(* IEC 61131-3 sources: rk/stdlib (part 4) *)

(* ---- Strings.st ---- *)
/*
String functions.

A `STRING` holds UTF-8 text, and its length is a number of bytes. The
functions here come in two families.

`LEN`, `FIND`, `LEFT`, `RIGHT`, `MID`, `INSERT`, `DELETE` and `REPLACE` count
bytes. They are the fast ones, and on ASCII text a byte is a character. On
other text a byte position can fall inside a character, and slicing there
yields a string that is not valid UTF-8.

The `CHAR_` functions count characters and never split one. A character is
one well-formed UTF-8 sequence. A byte that belongs to none counts as a
character on its own, its Latin-1 code point, like `CHAR#'$E9'`.

Positions start at 1 in both families. A function that returns a `STRING`
returns up to 255 bytes, and cuts a longer result there. It is also cut,
without an error, when it does not fit where it is stored.
*/
NAMESPACE Std.Strings

	/* Returns the length of `IN`, in bytes.

	   This is not the number of characters: `LEN('café')` is 5, because `é`
	   takes two bytes. See [Std.Strings.CHAR_COUNT] for that.

	   The length is stored with the string, so this does not scan it.

	   # Examples

	   ```iecst
	   n := LEN('hello');  // 5
	   n := LEN('');       // 0
	   ```
	*/
	FUNCTION LEN: UDINT
		VAR_INPUT
			IN: STRING[255];
		END_VAR
		{wasm 'str.byte_len' (params IN) (result LEN)}
	END_FUNCTION

	/* Returns `TRUE` if `IN` is well-formed UTF-8.

	   Text that comes from outside the program, such as a host import or a
	   fieldbus frame, may not be. Check it before slicing it by bytes.

	   # Examples

	   ```iecst
	   ok := IS_UTF8('café');  // TRUE
	   ok := IS_UTF8('$E9');   // FALSE, a lone Latin-1 byte
	   ```
	*/
	FUNCTION IS_UTF8: BOOL
		VAR_INPUT
			IN: STRING[255];
		END_VAR
		{wasm 'str.is_utf8' (params IN) (result IS_UTF8)}
	END_FUNCTION

	/* Returns the byte position of the first occurrence of `IN2` in
	   `IN1`, or 0 if there is none.

	   Positions start at 1. An empty `IN2` is found at position 1.

	   To look for a single `CHAR`, convert it with [Std.Convert.CHAR_TO_STRING].

	   # Examples

	   ```iecst
	   p := FIND('hello world', 'world');  // 7
	   p := FIND('hello world', 'xyz');    // 0
	   ```
	*/
	FUNCTION FIND: UDINT
		VAR_INPUT
			IN1: STRING[255];
			IN2: STRING[255];
		END_VAR
		{wasm 'str.byte_find' (params IN1 IN2) (result FIND)}
	END_FUNCTION

	/* Returns its inputs one after the other, from two inputs up to eight.

	   To append a single `CHAR`, convert it with [Std.Convert.CHAR_TO_STRING].

	   # Examples

	   ```iecst
	   s := CONCAT('hello ', 'world');  // 'hello world'
	   s := CONCAT('a', 'b', 'c');      // 'abc'
	   ```
	*/
	FUNCTION CONCAT: STRING[255]
		VAR_INPUT
			IN1: STRING[255];
			IN2: STRING[255];
		END_VAR
		{wasm 'str.concat' (params IN1 IN2) (result CONCAT)}
	END_FUNCTION

	FUNCTION CONCAT: STRING[255]
		VAR_INPUT
			IN1: STRING[255];
			IN2: STRING[255];
			IN3: STRING[255];
		END_VAR

		CONCAT := CONCAT(IN1, IN2);
		CONCAT := CONCAT(CONCAT, IN3);
	END_FUNCTION

	FUNCTION CONCAT: STRING[255]
		VAR_INPUT
			IN1: STRING[255];
			IN2: STRING[255];
			IN3: STRING[255];
			IN4: STRING[255];
		END_VAR

		CONCAT := CONCAT(IN1, IN2);
		CONCAT := CONCAT(CONCAT, IN3);
		CONCAT := CONCAT(CONCAT, IN4);
	END_FUNCTION

	FUNCTION CONCAT: STRING[255]
		VAR_INPUT
			IN1: STRING[255];
			IN2: STRING[255];
			IN3: STRING[255];
			IN4: STRING[255];
			IN5: STRING[255];
		END_VAR

		CONCAT := CONCAT(IN1, IN2);
		CONCAT := CONCAT(CONCAT, IN3);
		CONCAT := CONCAT(CONCAT, IN4);
		CONCAT := CONCAT(CONCAT, IN5);
	END_FUNCTION

	FUNCTION CONCAT: STRING[255]
		VAR_INPUT
			IN1: STRING[255];
			IN2: STRING[255];
			IN3: STRING[255];
			IN4: STRING[255];
			IN5: STRING[255];
			IN6: STRING[255];
		END_VAR

		CONCAT := CONCAT(IN1, IN2);
		CONCAT := CONCAT(CONCAT, IN3);
		CONCAT := CONCAT(CONCAT, IN4);
		CONCAT := CONCAT(CONCAT, IN5);
		CONCAT := CONCAT(CONCAT, IN6);
	END_FUNCTION

	FUNCTION CONCAT: STRING[255]
		VAR_INPUT
			IN1: STRING[255];
			IN2: STRING[255];
			IN3: STRING[255];
			IN4: STRING[255];
			IN5: STRING[255];
			IN6: STRING[255];
			IN7: STRING[255];
		END_VAR

		CONCAT := CONCAT(IN1, IN2);
		CONCAT := CONCAT(CONCAT, IN3);
		CONCAT := CONCAT(CONCAT, IN4);
		CONCAT := CONCAT(CONCAT, IN5);
		CONCAT := CONCAT(CONCAT, IN6);
		CONCAT := CONCAT(CONCAT, IN7);
	END_FUNCTION

	FUNCTION CONCAT: STRING[255]
		VAR_INPUT
			IN1: STRING[255];
			IN2: STRING[255];
			IN3: STRING[255];
			IN4: STRING[255];
			IN5: STRING[255];
			IN6: STRING[255];
			IN7: STRING[255];
			IN8: STRING[255];
		END_VAR

		CONCAT := CONCAT(IN1, IN2);
		CONCAT := CONCAT(CONCAT, IN3);
		CONCAT := CONCAT(CONCAT, IN4);
		CONCAT := CONCAT(CONCAT, IN5);
		CONCAT := CONCAT(CONCAT, IN6);
		CONCAT := CONCAT(CONCAT, IN7);
		CONCAT := CONCAT(CONCAT, IN8);
	END_FUNCTION

	/* Returns the first `L` bytes of `IN`.

	   Returns all of `IN` when `L` is greater than its length.

	   # Examples

	   ```iecst
	   s := LEFT('hello world', 5);  // 'hello'
	   s := LEFT('hi', 10);          // 'hi'
	   ```
	*/
	FUNCTION LEFT: STRING[255]
		VAR_INPUT
			IN: STRING[255];
			L: UDINT;
		END_VAR
		{wasm 'str.byte_left' (params IN L) (result LEFT)}
	END_FUNCTION

	/* Returns the last `L` bytes of `IN`.

	   Returns all of `IN` when `L` is greater than its length.

	   # Examples

	   ```iecst
	   s := RIGHT('hello world', 5);  // 'world'
	   s := RIGHT('hi', 10);          // 'hi'
	   ```
	*/
	FUNCTION RIGHT: STRING[255]
		VAR_INPUT
			IN: STRING[255];
			L: UDINT;
		END_VAR
		{wasm 'str.byte_right' (params IN L) (result RIGHT)}
	END_FUNCTION

	/* Returns `L` bytes of `IN`, starting at byte position `P`.

	   Returns fewer when `IN` ends first, and an empty string when `P` is 0 or
	   past the end.

	   # Examples

	   ```iecst
	   s := MID('hello world', 5, 7);  // 'world'
	   s := MID('hello', 10, 3);       // 'llo'
	   s := MID('hello', 3, 10);       // ''
	   ```
	*/
	FUNCTION MID: STRING[255]
		VAR_INPUT
			IN: STRING[255];
			L: UDINT;
			P: UDINT;
		END_VAR
		{wasm 'str.byte_mid' (params IN L P) (result MID)}
	END_FUNCTION

	/* Returns `IN1` with `IN2` inserted after byte position `P`.

	   A `P` of 0 inserts at the front.

	   To insert a single `CHAR`, convert it with [Std.Convert.CHAR_TO_STRING].

	   # Examples

	   ```iecst
	   s := INSERT('helloworld', 'XX', 5);  // 'helloXXworld'
	   s := INSERT('world', 'hello ', 0);   // 'hello world'
	   ```
	*/
	FUNCTION INSERT: STRING[255]
		VAR_INPUT
			IN1: STRING[255];
			IN2: STRING[255];
			P: UDINT;
		END_VAR
		{wasm 'str.byte_insert' (params IN1 IN2 P) (result INSERT)}
	END_FUNCTION

	/* Returns `IN` without the `L` bytes that start at byte position `P`.

	   Removes fewer when `IN` ends first, and nothing when `P` is past the end.

	   # Examples

	   ```iecst
	   s := DELETE('hello world', 6, 6);  // 'hello'
	   s := DELETE('hello', 10, 3);       // 'he'
	   s := DELETE('hello', 3, 10);       // 'hello'
	   ```
	*/
	FUNCTION DELETE: STRING[255]
		VAR_INPUT
			IN: STRING[255];
			L: UDINT;
			P: UDINT;
		END_VAR
		{wasm 'str.byte_delete' (params IN L P) (result DELETE)}
	END_FUNCTION

	/* Returns `IN1` with the `L` bytes that start at byte position `P` replaced
	   by `IN2`.

	   `IN2` does not have to be `L` bytes long.

	   To replace with a single `CHAR`, convert it with [Std.Convert.CHAR_TO_STRING].

	   # Examples

	   ```iecst
	   s := REPLACE('hello world', 'there', 5, 7);  // 'hello there'
	   s := REPLACE('hello world', '!', 5, 7);      // 'hello !'
	   ```
	*/
	FUNCTION REPLACE: STRING[255]
		VAR_INPUT
			IN1: STRING[255];
			IN2: STRING[255];
			L: UDINT;
			P: UDINT;
		END_VAR
		{wasm 'str.byte_replace' (params IN1 IN2 L P) (result REPLACE)}
	END_FUNCTION

	/* Returns the number of characters in `IN`.

	   # Examples

	   ```iecst
	   n := CHAR_COUNT('café');    // 4, where LEN returns 5
	   n := CHAR_COUNT('日本語');  // 3, where LEN returns 9
	   ```
	*/
	FUNCTION CHAR_COUNT: UDINT
		VAR_INPUT
			IN: STRING[255];
		END_VAR
		{wasm 'str.char_count' (params IN) (result CHAR_COUNT)}
	END_FUNCTION

	/* Returns the character at position `P` of `IN`.

	   Returns `CHAR#'$00'` when `P` is 0 or past the end.

	   # Examples

	   ```iecst
	   c := CHAR_AT('café', 4);  // CHAR#'é'
	   c := CHAR_AT('abc', 4);   // CHAR#'$00'
	   ```
	*/
	FUNCTION CHAR_AT: CHAR
		VAR_INPUT
			IN: STRING[255];
			P: UDINT;
		END_VAR
		{wasm 'str.char_at' (params IN P) (result CHAR_AT)}
	END_FUNCTION

	/* Returns the character position of the first occurrence of `IN2` in
	   `IN1`, or 0 if there is none.

	   An empty `IN2` is found at position 1, as with [Std.Strings.FIND].

	   # Examples

	   ```iecst
	   p := CHAR_FIND('日本語', '語');  // 3, where FIND returns 7
	   p := CHAR_FIND('abc', 'x');      // 0
	   ```
	*/
	FUNCTION CHAR_FIND: UDINT
		VAR_INPUT
			IN1: STRING[255];
			IN2: STRING[255];
		END_VAR
		{wasm 'str.char_find' (params IN1 IN2) (result CHAR_FIND)}
	END_FUNCTION

	/* Returns the first `L` characters of `IN`.

	   Returns all of `IN` when `L` is greater than its character count.

	   # Examples

	   ```iecst
	   s := CHAR_LEFT('café', 3);   // 'caf'
	   s := CHAR_LEFT('café', 10);  // 'café'
	   ```
	*/
	FUNCTION CHAR_LEFT: STRING[255]
		VAR_INPUT
			IN: STRING[255];
			L: UDINT;
		END_VAR
		{wasm 'str.char_left' (params IN L) (result CHAR_LEFT)}
	END_FUNCTION

	/* Returns the last `L` characters of `IN`.

	   Returns all of `IN` when `L` is greater than its character count.

	   # Examples

	   ```iecst
	   s := CHAR_RIGHT('日本語', 2);  // '本語'
	   s := CHAR_RIGHT('café', 1);    // 'é'
	   ```
	*/
	FUNCTION CHAR_RIGHT: STRING[255]
		VAR_INPUT
			IN: STRING[255];
			L: UDINT;
		END_VAR
		{wasm 'str.char_right' (params IN L) (result CHAR_RIGHT)}
	END_FUNCTION

	/* Returns `L` characters of `IN`, starting at character position `P`.

	   Returns fewer when `IN` ends first, and an empty string when `P` is 0 or
	   past the end.

	   # Examples

	   ```iecst
	   s := CHAR_MID('café', 2, 3);    // 'fé'
	   s := CHAR_MID('日本語', 1, 2);  // '本'
	   ```
	*/
	FUNCTION CHAR_MID: STRING[255]
		VAR_INPUT
			IN: STRING[255];
			L: UDINT;
			P: UDINT;
		END_VAR
		{wasm 'str.char_mid' (params IN L P) (result CHAR_MID)}
	END_FUNCTION

	/* Returns `IN1` with `IN2` inserted after character position `P`.

	   A `P` of 0 inserts at the front, and a `P` past the end appends.

	   # Examples

	   ```iecst
	   s := CHAR_INSERT('caf', 'é', 3);    // 'café'
	   s := CHAR_INSERT('abc', 'X', 0);    // 'Xabc'
	   s := CHAR_INSERT('café', 'X', 99);  // 'caféX'
	   ```
	*/
	FUNCTION CHAR_INSERT: STRING[255]
		VAR_INPUT
			IN1: STRING[255];
			IN2: STRING[255];
			P: UDINT;
		END_VAR
		{wasm 'str.char_insert' (params IN1 IN2 P) (result CHAR_INSERT)}
	END_FUNCTION

	/* Returns `IN` without the `L` characters that start at character
	   position `P`.

	   Returns `IN` unchanged when `P` is 0 or past the end.

	   # Examples

	   ```iecst
	   s := CHAR_DELETE('日本語', 1, 2);  // '日語'
	   s := CHAR_DELETE('café', 1, 5);    // 'café'
	   ```
	*/
	FUNCTION CHAR_DELETE: STRING[255]
		VAR_INPUT
			IN: STRING[255];
			L: UDINT;
			P: UDINT;
		END_VAR
		{wasm 'str.char_delete' (params IN L P) (result CHAR_DELETE)}
	END_FUNCTION

	/* Returns `IN1` with the `L` characters that start at character position
	   `P` replaced by `IN2`.

	   Returns `IN1` unchanged when `P` is 0 or past the end.

	   # Examples

	   ```iecst
	   s := CHAR_REPLACE('café', 'e', 1, 4);    // 'cafe'
	   s := CHAR_REPLACE('日本語', 'X', 2, 1);  // 'X語'
	   ```
	*/
	FUNCTION CHAR_REPLACE: STRING[255]
		VAR_INPUT
			IN1: STRING[255];
			IN2: STRING[255];
			L: UDINT;
			P: UDINT;
		END_VAR
		{wasm 'str.char_replace' (params IN1 IN2 L P) (result CHAR_REPLACE)}
	END_FUNCTION

	NAMESPACE Test
		USING Std.Unit
		USING Std.Convert

		{test}
		FUNCTION test_len_ascii
			ASSERT(LEN('hello') = 5);
		END_FUNCTION

		{test}
		FUNCTION test_len_empty
			ASSERT(LEN('') = 0);
		END_FUNCTION

		{test}
		FUNCTION test_len_counts_utf8_bytes
			ASSERT(LEN('café') = 5 AND LEN('€') = 3 AND LEN('中文') = 6);
			ASSERT(IS_UTF8('café') AND IS_UTF8('中文'));
			{allow 'latin1-escape'}
			ASSERT(LEN('$E9') = 1 AND NOT IS_UTF8('$E9'));
		END_FUNCTION

		{test}
		FUNCTION test_is_utf8_ascii
			ASSERT(IS_UTF8('hello'));
		END_FUNCTION

		{test}
		FUNCTION test_is_utf8_empty
			ASSERT(IS_UTF8(''));
		END_FUNCTION

		{test}
		FUNCTION test_find_present
			ASSERT(FIND('hello world', 'world') = 7);
		END_FUNCTION

		{test}
		FUNCTION test_find_at_start
			ASSERT(FIND('hello world', 'hello') = 1);
		END_FUNCTION

		{test}
		FUNCTION test_find_missing
			ASSERT(FIND('hello world', 'xyz') = 0);
		END_FUNCTION

		{test}
		FUNCTION test_find_empty_needle
			ASSERT(FIND('hello', '') = 1);
		END_FUNCTION

		{test}
		FUNCTION test_find_needle_longer_than_haystack
			ASSERT(FIND('hi', 'hello') = 0);
		END_FUNCTION

		{test}
		FUNCTION test_concat_basic
			VAR result: STRING; END_VAR
			result := CONCAT('hello ', 'world');
			ASSERT(LEN(result) = 11);
			ASSERT(FIND(result, 'hello world') = 1);
		END_FUNCTION

		{test}
		FUNCTION test_concat_empty_left
			VAR result: STRING; END_VAR
			result := CONCAT('', 'world');
			ASSERT(LEN(result) = 5);
		END_FUNCTION

		{test}
		FUNCTION test_concat_empty_right
			VAR result: STRING; END_VAR
			result := CONCAT('hello', '');
			ASSERT(LEN(result) = 5);
		END_FUNCTION

		// A result holds up to 255 bytes, not the default 80: what does not
		// fit is cut where it is stored.
		{test}
		FUNCTION test_concat_keeps_more_than_80_bytes
			VAR
				a: STRING[100] := '0123456789012345678901234567890123456789012345678901234567890123456789012345678901234567890123456789';
				result: STRING[200];
			END_VAR
			result := CONCAT(a, a);
			ASSERT(LEN(result) = 200);
		END_FUNCTION

		{test}
		FUNCTION test_a_result_is_cut_at_255_bytes
			VAR
				a: STRING[200] := '01234567890123456789012345678901234567890123456789012345678901234567890123456789012345678901234567890123456789012345678901234567890123456789012345678901234567890123456789012345678901234567890123456789';
				result: STRING[300];
			END_VAR
			result := CONCAT(a, a);
			// LEN reads 255 bytes at most: the result holds 255.
			{allow 'string-truncation'}
			ASSERT(LEN(result) = 255);
		END_FUNCTION

		{test}
		FUNCTION test_delete_one_byte_of_a_100_byte_string
			VAR s: STRING[200] := '0123456789012345678901234567890123456789012345678901234567890123456789012345678901234567890123456789'; END_VAR
			s := DELETE(s, 1, 1);
			ASSERT(LEN(s) = 99);
		END_FUNCTION

		{test}
		FUNCTION test_left_basic
			VAR result: STRING; END_VAR
			result := LEFT('hello world', 5);
			ASSERT(LEN(result) = 5);
			ASSERT(FIND(result, 'hello') = 1);
		END_FUNCTION

		{test}
		FUNCTION test_left_n_exceeds_length
			VAR result: STRING; END_VAR
			result := LEFT('hi', 10);
			ASSERT(LEN(result) = 2);
		END_FUNCTION

		{test}
		FUNCTION test_right_basic
			VAR result: STRING; END_VAR
			result := RIGHT('hello world', 5);
			ASSERT(LEN(result) = 5);
			ASSERT(FIND(result, 'world') = 1);
		END_FUNCTION

		{test}
		FUNCTION test_mid_basic
			VAR result: STRING; END_VAR
			// 'world' starts at byte 7, 5 chars
			result := MID('hello world', 5, 7);
			ASSERT(LEN(result) = 5);
			ASSERT(FIND(result, 'world') = 1);
		END_FUNCTION

		{test}
		FUNCTION test_mid_p_zero
			VAR result: STRING; END_VAR
			result := MID('hello', 3, 0);
			ASSERT(LEN(result) = 0);
		END_FUNCTION

		{test}
		FUNCTION test_insert_middle
			VAR result: STRING; END_VAR
			// Insert 'XX' after byte 5 of 'helloworld' → 'helloXXworld'
			result := INSERT('helloworld', 'XX', 5);
			ASSERT(LEN(result) = 12);
			ASSERT(FIND(result, 'helloXXworld') = 1);
		END_FUNCTION

		{test}
		FUNCTION test_insert_front
			VAR result: STRING; END_VAR
			result := INSERT('world', 'hello ', 0);
			ASSERT(LEN(result) = 11);
			ASSERT(FIND(result, 'hello world') = 1);
		END_FUNCTION

		{test}
		FUNCTION test_delete_basic
			VAR result: STRING; END_VAR
			// Delete 6 bytes starting at byte 6 of 'hello world' → 'hello'
			result := DELETE('hello world', 6, 6);
			ASSERT(LEN(result) = 5);
			ASSERT(FIND(result, 'hello') = 1);
		END_FUNCTION

		{test}
		FUNCTION test_replace_basic
			VAR result: STRING; END_VAR
			// Replace 5 bytes at byte 7 of 'hello world' with 'there'
			result := REPLACE('hello world', 'there', 5, 7);
			ASSERT(LEN(result) = 11);
			ASSERT(FIND(result, 'hello there') = 1);
		END_FUNCTION

		{test}
		FUNCTION test_concat_nested_binary
			// Independent inner CONCATs feeding an outer CONCAT: each
			// inner result must survive long enough for the outer to read
			// it. With per-call-site scratch slots: 'xxyyzzww'.
			VAR result: STRING; END_VAR
			result := CONCAT(CONCAT('xx', 'yy'), CONCAT('zz', 'ww'));
			ASSERT(LEN(result) = 8);
			ASSERT(FIND(result, 'xxyyzzww') = 1);
		END_FUNCTION

		{test}
		FUNCTION test_concat_nested_left_arg
			// Inner result used as outer's first arg.
			VAR result: STRING; END_VAR
			result := CONCAT(CONCAT('ab', 'cd'), 'ef');
			ASSERT(LEN(result) = 6);
			ASSERT(FIND(result, 'abcdef') = 1);
		END_FUNCTION

		{test}
		FUNCTION test_left_inside_concat
			VAR result: STRING; END_VAR
			result := CONCAT(LEFT('hello world', 5), '!');
			ASSERT(LEN(result) = 6);
			ASSERT(FIND(result, 'hello!') = 1);
		END_FUNCTION

		/* CHAR-as-string usage: explicit conversion via
		   `Std.Convert.CHAR_TO_STRING`. CHAR is an i32 code point at
		   the WASM ABI; CONCAT/INSERT/REPLACE/FIND all take STRING args,
		   so users wrap CHAR values explicitly. */

		{test}
		FUNCTION test_concat_char_literal_right
			VAR result: STRING; END_VAR
			result := CONCAT('hello', CHAR_TO_STRING(CHAR#'!'));
			ASSERT(LEN(result) = 6);
			ASSERT(FIND(result, 'hello!') = 1);
		END_FUNCTION

		{test}
		FUNCTION test_concat_char_literal_left
			VAR result: STRING; END_VAR
			result := CONCAT(CHAR_TO_STRING(CHAR#'>'), ' message');
			ASSERT(LEN(result) = 9);
			ASSERT(FIND(result, '> message') = 1);
		END_FUNCTION

		{test}
		FUNCTION test_find_char_literal_needle
			ASSERT(FIND('hello', CHAR_TO_STRING(CHAR#'l')) = 3);
		END_FUNCTION

		{test}
		FUNCTION test_insert_char_literal
			VAR result: STRING; END_VAR
			result := INSERT('helloworld', CHAR_TO_STRING(CHAR#' '), 5);
			ASSERT(LEN(result) = 11);
			ASSERT(FIND(result, 'hello world') = 1);
		END_FUNCTION

		{test}
		FUNCTION test_replace_char_literal
			VAR result: STRING; END_VAR
			// Replace 5 bytes at byte 7 of 'hello world' with the single CHAR '!'.
			result := REPLACE('hello world', CHAR_TO_STRING(CHAR#'!'), 5, 7);
			ASSERT(LEN(result) = 7);
			ASSERT(FIND(result, 'hello !') = 1);
		END_FUNCTION

		{test}
		FUNCTION test_concat_char_var
			VAR
				bang: CHAR := CHAR#'!';
				result: STRING;
			END_VAR
			result := CONCAT('hello', CHAR_TO_STRING(bang));
			ASSERT(LEN(result) = 6);
			ASSERT(FIND(result, 'hello!') = 1);
		END_FUNCTION

		{test}
		FUNCTION test_find_char_var
			VAR
				needle: CHAR := CHAR#'l';
			END_VAR
			ASSERT(FIND('hello', CHAR_TO_STRING(needle)) = 3);
		END_FUNCTION

		{test}
		FUNCTION test_concat_char_var_left
			VAR
				prefix: CHAR := CHAR#'>';
				result: STRING;
			END_VAR
			result := CONCAT(CHAR_TO_STRING(prefix), ' message');
			ASSERT(LEN(result) = 9);
			ASSERT(FIND(result, '> message') = 1);
		END_FUNCTION

		{test}
		FUNCTION test_concat_two_char_vars
			// Two nested CHAR_TO_STRING calls: each must get its own
			// per-call-site scratch slot, the second mustn't clobber the
			// first before the outer CONCAT reads them.
			VAR
				a: CHAR := CHAR#'a';
				b: CHAR := CHAR#'b';
				result: STRING;
			END_VAR
			result := CONCAT(CHAR_TO_STRING(a), CHAR_TO_STRING(b));
			ASSERT(LEN(result) = 2);
			ASSERT(FIND(result, 'ab') = 1);
		END_FUNCTION

		// --- return-slot aliasing: results copied into locals must survive
		// LATER producer calls (the dangerous scenario of a shared static
		// return slot), and self-argument accumulation must not corrupt ---

		{test}
		FUNCTION test_result_survives_later_producer_call
			VAR
				first, second: STRING;
			END_VAR
			first := CONCAT('aa', 'bb');
			second := CONCAT('cc', 'dd');
			ASSERT(FIND(first, 'aabb') = 1, 'earlier result must survive a later producer call');
			ASSERT(FIND(second, 'ccdd') = 1, 'later result is correct too');
		END_FUNCTION

		{test}
		FUNCTION test_concat_self_accumulation
			VAR
				s: STRING;
				i: INT;
			END_VAR
			s := 'x';
			FOR i := 1 TO 4 DO
				s := CONCAT(s, 'y');
			END_FOR;
			ASSERT(LEN(s) = 5, 'x + 4 accumulated y');
			ASSERT(FIND(s, 'xyyyy') = 1, 'self-argument CONCAT accumulates correctly');
		END_FUNCTION

		// --- slicer bounds: N/P beyond the string must clamp, not underflow ---

		{test}
		FUNCTION test_right_n_beyond_length
			VAR
				s: STRING;
			END_VAR
			// RIGHT computes len-N internally: N > len must clamp, not
			// underflow to a huge unsigned offset.
			s := RIGHT('hi', 10);
			ASSERT(LEN(s) = 2, 'RIGHT with N beyond length returns the whole string');
			ASSERT(FIND(s, 'hi') = 1, 'content intact');
		END_FUNCTION

		{test}
		FUNCTION test_mid_beyond_length
			VAR
				s: STRING;
			END_VAR
			s := MID('hello', 10, 3);
			ASSERT(LEN(s) = 3, 'MID clamps L to the remaining chars');
			s := MID('hello', 3, 10);
			ASSERT(LEN(s) = 0, 'MID with P beyond length yields empty');
		END_FUNCTION

		{test}
		FUNCTION test_delete_beyond_length
			VAR
				s: STRING;
			END_VAR
			// Signature is DELETE(S, N, P): delete N chars at position P.
			s := DELETE('hello', 3, 10);
			ASSERT(LEN(s) = 5, 'DELETE at P beyond the end removes nothing');
			s := DELETE('hello', 10, 3);
			ASSERT(LEN(s) = 2, 'DELETE clamps N to the remaining chars (keeps "he")');
			ASSERT(FIND(s, 'he') = 1, 'prefix before P survives');
		END_FUNCTION

		{test}
		FUNCTION test_find_no_match_returns_zero
			ASSERT(FIND('hello', 'xyz') = 0, 'FIND with no match returns 0');
			ASSERT(FIND('', 'a') = 0, 'FIND in empty string returns 0');
		END_FUNCTION

		{test}
		FUNCTION test_len_zero_slices
			VAR
				s: STRING;
			END_VAR
			s := LEFT('hello', 0);
			ASSERT(LEN(s) = 0, 'LEFT L=0 is empty');
			s := MID('hello', 0, 2);
			ASSERT(LEN(s) = 0, 'MID L=0 is empty');
		END_FUNCTION

		// --- STRING comparison operators: =, <>, and lexicographic ordering
		// (byte-wise with length tiebreak). These replace the LEN+FIND idiom
		// for content assertions. ---

		{test}
		FUNCTION test_string_equality_operators
			VAR
				s: STRING := 'START';
			END_VAR
			ASSERT(s = 'START', 'var = literal');
			ASSERT('START' = s, 'literal = var');
			ASSERT(s <> 'STOP', 'not-equal');
			ASSERT_EQ(CONCAT('STA', 'RT'), 'START', 'ASSERT_EQ on a producer result');
			ASSERT_NEQ(CONCAT('a', 'b'), 'ba', 'ASSERT_NEQ on unequal content');
		END_FUNCTION

		{test}
		FUNCTION test_string_ordering_operators
			ASSERT('abc' < 'abd', 'lexicographic less');
			ASSERT('ab' < 'abc', 'shared prefix: shorter is smaller');
			ASSERT('abd' > 'abc', 'greater');
			ASSERT('abc' <= 'abc', 'le on equal');
			ASSERT('abc' >= 'abc', 'ge on equal');
			ASSERT(NOT ('abc' < 'abc'), 'not strictly less than itself');
			ASSERT('' < 'a', 'empty sorts first');
		END_FUNCTION

		{test}
		FUNCTION test_string_equality_after_mutation
			VAR
				s: STRING := 'x';
				i: INT;
			END_VAR
			FOR i := 1 TO 3 DO
				s := CONCAT(s, 'y');
			END_FOR;
			ASSERT_EQ(s, 'xyyy', 'accumulated content compares whole');
		END_FUNCTION

		// Both operands are producer calls: each needs its own scratch
		// buffer. If they shared the one static return slot, the second call
		// would clobber the first and every such comparison would degenerate
		// to comparing a value with itself (silently always equal).
		{test}
		FUNCTION test_string_comparison_between_two_producers
			ASSERT(CONCAT('ab', 'cd') = CONCAT('ab', 'cd'), 'equal producer results compare equal');
			ASSERT(CONCAT('ab', 'cd') <> CONCAT('xy', 'zw'), 'different producer results must not be equal');
			ASSERT(CONCAT('a', 'a') < CONCAT('a', 'b'), 'ordering holds across two producers');
		END_FUNCTION

		// ----- Character-aware twins --------------------------------------
		{test}
		FUNCTION test_char_count_agrees_with_len_on_ascii
			ASSERT(CHAR_COUNT('hello') = 5 AND CHAR_COUNT('') = 0);
			ASSERT(CHAR_COUNT('hello') = LEN('hello'));
		END_FUNCTION

		{test}
		FUNCTION test_char_count_counts_characters_not_bytes
			ASSERT(CHAR_COUNT('café') = 4 AND LEN('café') = 5);
			ASSERT(CHAR_COUNT('日本語') = 3 AND LEN('日本語') = 9);
			{allow 'latin1-escape'}
			ASSERT(CHAR_COUNT('$E9$E9') = 2, 'a stray byte is one character');
		END_FUNCTION

		{test}
		FUNCTION test_char_at_returns_the_character
			ASSERT(CHAR_AT('café', 4) = CHAR#'é' AND CHAR_AT('café', 1) = CHAR#'c');
			ASSERT(CHAR_AT('日本語', 2) = CHAR#'本');
			{allow 'latin1-escape'}
			ASSERT(CHAR_AT('$E9', 1) = CHAR#'é', 'a stray byte reads as its Latin-1 character');
			ASSERT(CHAR_AT('abc', 0) = CHAR#'$00' AND CHAR_AT('abc', 4) = CHAR#'$00');
		END_FUNCTION

		{test}
		FUNCTION test_char_find_counts_characters
			ASSERT(CHAR_FIND('日本語', '語') = 3 AND FIND('日本語', '語') = 7);
			ASSERT(CHAR_FIND('café!', '!') = 5);
			ASSERT(CHAR_FIND('abc', 'x') = 0 AND CHAR_FIND('abc', '') = 1);
		END_FUNCTION

		{test}
		FUNCTION test_char_left_and_right_never_split_a_character
			ASSERT(CHAR_LEFT('café', 4) = 'café' AND CHAR_LEFT('café', 3) = 'caf');
			ASSERT(CHAR_RIGHT('café', 1) = 'é' AND CHAR_RIGHT('日本語', 2) = '本語');
			ASSERT(CHAR_LEFT('café', 10) = 'café' AND CHAR_RIGHT('café', 0) = '');
		END_FUNCTION

		{test}
		FUNCTION test_char_mid_counts_characters
			ASSERT(CHAR_MID('日本語', 1, 2) = '本' AND CHAR_MID('café', 2, 3) = 'fé');
			ASSERT(CHAR_MID('café', 10, 4) = 'é', 'N past the end is clamped');
			ASSERT(CHAR_MID('café', 1, 0) = '' AND CHAR_MID('café', 1, 5) = '');
		END_FUNCTION

		{test}
		FUNCTION test_char_insert_delete_replace_count_characters
			ASSERT(CHAR_INSERT('caf', 'é', 3) = 'café' AND CHAR_INSERT('日語', '本', 1) = '日本語');
			ASSERT(CHAR_INSERT('abc', 'X', 0) = 'Xabc');
			ASSERT(CHAR_DELETE('café', 1, 4) = 'caf' AND CHAR_DELETE('日本語', 1, 2) = '日語');
			ASSERT(CHAR_DELETE('café', 1, 0) = 'café' AND CHAR_DELETE('café', 1, 5) = 'café');
			ASSERT(CHAR_REPLACE('café', 'e', 1, 4) = 'cafe' AND CHAR_REPLACE('日本語', 'X', 2, 1) = 'X語');
			ASSERT(CHAR_REPLACE('café', 'X', 1, 0) = 'café');
		END_FUNCTION

		// A character position past the end maps to a byte position past the
		// end and the byte functions decide: just past and far past must agree.
		{test}
		FUNCTION test_char_positions_past_the_end_agree
			ASSERT(CHAR_MID('café', 2, 5) = CHAR_MID('café', 2, 99) AND CHAR_MID('café', 2, 99) = '');
			ASSERT(CHAR_DELETE('café', 2, 5) = CHAR_DELETE('café', 2, 99) AND CHAR_DELETE('café', 2, 99) = 'café');
			ASSERT(CHAR_REPLACE('café', 'X', 2, 5) = CHAR_REPLACE('café', 'X', 2, 99) AND CHAR_REPLACE('café', 'X', 2, 99) = 'café');
			ASSERT(CHAR_INSERT('café', 'X', 5) = CHAR_INSERT('café', 'X', 99) AND CHAR_INSERT('café', 'X', 99) = 'caféX');
		END_FUNCTION

		// `LEN(s) - k` with k > LEN(s) is an N near 2^32, and `start + n`
		// wrapped on wasm32: MID trapped, DELETE and REPLACE kept the wrong
		// part. CHAR_MID and its kin count N first and never did.
		{test}
		FUNCTION test_mid_delete_replace_with_n_near_the_limit
			ASSERT(MID('hello', UDINT#4294967295, 2) = 'ello', 'MID N = 2^32-1');
			ASSERT(MID('hello', UDINT#4294967294, 3) = 'llo', 'MID N = 2^32-2 at P = 3');
			ASSERT(DELETE('hello', UDINT#4294967295, 3) = 'he', 'DELETE N = 2^32-1');
			ASSERT(REPLACE('hello', 'Y', UDINT#4294967295, 3) = 'heY', 'REPLACE N = 2^32-1');
			ASSERT(CHAR_MID('café', UDINT#4294967295, 2) = 'afé', 'CHAR_MID N = 2^32-1');
			ASSERT(CHAR_DELETE('café', UDINT#4294967295, 2) = 'c', 'CHAR_DELETE N = 2^32-1');
			ASSERT(CHAR_REPLACE('café', 'X', UDINT#4294967295, 2) = 'cX', 'CHAR_REPLACE N = 2^32-1');
		END_FUNCTION

		{test}
		FUNCTION test_n_from_len_minus_k_past_the_end
			VAR s : STRING := 'hello'; k : UDINT := 7; END_VAR
			ASSERT(MID(s, LEN(s) - k, 2) = 'ello', 'MID with LEN(s) - k');
			ASSERT(DELETE(s, LEN(s) - k, 2) = 'h', 'DELETE with LEN(s) - k');
			ASSERT(REPLACE(s, '-', LEN(s) - k, 2) = 'h-', 'REPLACE with LEN(s) - k');
		END_FUNCTION

		{test}
		FUNCTION test_insert_past_the_end_appends
			ASSERT(INSERT('hello', 'X', 6) = 'helloX', 'P = LEN + 1');
			ASSERT(INSERT('hello', 'X', UDINT#4294967295) = 'helloX', 'P = 2^32-1');
			ASSERT(INSERT('', 'X', 0) = 'X', 'into an empty string');
		END_FUNCTION

		{test}
		FUNCTION test_replace_with_an_empty_ins_deletes
			ASSERT(REPLACE('hello', '', 2, 2) = 'hlo', 'an empty INS');
			ASSERT(REPLACE('hello', 'X', 0, 3) = 'heXllo', 'N = 0 inserts');
		END_FUNCTION

		{test}
		FUNCTION test_find_on_empty_strings
			ASSERT(FIND('', 'a') = 0, 'an empty haystack');
			ASSERT(FIND('', '') = 1, 'both empty');
			ASSERT(CHAR_FIND('café', '') = 1, 'an empty needle');
		END_FUNCTION
	END_NAMESPACE

END_NAMESPACE

(* ---- Timers.st ---- *)
/*
Timers, and the clocks they read.

Each takes `IN` and a duration `PT`, and gives `Q` and the elapsed time
`ET`, which stops at `PT`. They read the clock when they are called, so a
timer is as precise as the scan that calls it.

`TP`, `TON` and `TOF` measure in `TIME`. The `_LTIME` blocks are the same
timers in `LTIME`.

`PLC_TIME` and `PLC_LTIME` read the monotonic clock, for the time between
two readings. `WALL_LDT`, `WALL_DT`, `LOCAL_LDT` and `LOCAL_OFFSET` read
the wall clock and the host's zone. The wall clock goes back when the
host's clock is set: a duration is measured with `PLC_TIME`.

A timer decides on `CURRENT_TIME - START_TIME`, a difference, which wraps
with the clock where `START_TIME + PT` would not: the host picks where the
monotonic clock starts, and `PLC_TIME` cycles every 49.7 days in any case.

A timer's step and clock readings are `NON_RETAIN`: held by a retained
instance, it starts over after a warm start instead of measuring from a
reading of the previous run's clock. `Q` and `ET` follow the step on every
call, so the first call after the warm start ends what the step no longer
runs.
*/
NAMESPACE Std.Timers
	USING Std.Convert;

	/* Returns the host's monotonic clock, which never goes back.

	   This is the `now` of the WASI
	   [monotonic clock](https://github.com/WebAssembly/WASI/blob/main/proposals/clocks/README.md),
	   a count of nanoseconds, and the one import a module that uses a timer
	   has.
	*/
	FUNCTION PRIVATE MONOTONIC_LTIME: LTIME
		MONOTONIC_LTIME := LINT_TO_LTIME(ULINT_TO_LINT(Wasi.Clocks.MonotonicClock.NOW()));
	END_FUNCTION

	/* Returns the monotonic clock as a `TIME`. Only the difference between two readings means something. */
	FUNCTION PLC_TIME: TIME
		PLC_TIME := LTIME_TO_TIME(MONOTONIC_LTIME());
	END_FUNCTION

	/* Returns the monotonic clock as an `LTIME`. Only the difference between two readings means something. */
	FUNCTION PLC_LTIME: LTIME
		PLC_LTIME := MONOTONIC_LTIME();
	END_FUNCTION

	/* Returns the host's wall clock as an `LDT`, in UTC: the `now` of the
	   WASI [system clock](https://github.com/WebAssembly/WASI/blob/main/proposals/clocks/README.md),
	   the seconds since 1970-01-01, negative before, and the nanoseconds
	   after them. */
	FUNCTION WALL_LDT : LDT
		VAR
			instant : Wasi.Clocks.SystemClock.INSTANT;
		END_VAR
		instant := Wasi.Clocks.SystemClock.NOW();
		WALL_LDT := LINT_TO_LDT(instant.seconds * LINT#1000000000 + instant.nanoseconds);
	END_FUNCTION

	/* Returns the host's wall clock as a `DT`, in UTC. */
	FUNCTION WALL_DT : DT
		WALL_DT := LDT_TO_DT(WALL_LDT());
	END_FUNCTION

	/* Returns how far east of UTC the host's zone is at `IN`, daylight
	   saving included: `LT#1h` in Paris in winter, `LT#2h` in summer,
	   `LT#-5h` in New York in winter. Raises "the host has no time zone"
	   when the host has none.

	   The zone is WASI 0.3's `timezone`, which is still unstable
	   (`clocks-timezone`): a host has it only with that feature on, and
	   its signature can change in a 0.3 release. */
	{warn = 'reads the time zone, which WASI 0.3 marks unstable: a host has it only with its clocks-timezone feature on'}
	FUNCTION LOCAL_OFFSET : LTIME
		VAR_INPUT
			IN : LDT;
		END_VAR
		VAR
			when : Wasi.Clocks.SystemClock.INSTANT;
			nanoseconds : LINT;
			known : BOOL;
			offset : LINT;
		END_VAR
		// WASI takes the whole seconds, rounded down, and the nanoseconds after them.
		when.seconds := LDT_TO_LINT(IN) / LINT#1000000000;
		nanoseconds := LDT_TO_LINT(IN) MOD LINT#1000000000;
		IF nanoseconds < LINT#0 THEN
			when.seconds := when.seconds - LINT#1;
			nanoseconds := nanoseconds + LINT#1000000000;
		END_IF;
		when.nanoseconds := LINT_TO_UDINT(nanoseconds);
		// The `utc-offset` of the WASI time zone: an `option<s64>`, which
		// comes back as whether the host has a zone, then the offset.
		Wasi.Clocks.Timezone.UTC_OFFSET(when := when, is_some => known, value => offset);
		IF NOT known THEN
			__RAISE('the host has no time zone');
		END_IF;
		LOCAL_OFFSET := LINT_TO_LTIME(offset);
	END_FUNCTION

	/* Returns the host's wall clock as an `LDT` in the host's zone: the
	   instant `WALL_LDT` returns, shifted by `LOCAL_OFFSET`, in the same
	   encoding. What a clock on the wall shows. Raises "the host has no
	   time zone" when the host has none, as `LOCAL_OFFSET` does. */
	{warn = 'reads the time zone, which WASI 0.3 marks unstable: a host has it only with its clocks-timezone feature on'}
	FUNCTION LOCAL_LDT : LDT
		VAR
			utc : LDT;
		END_VAR
		utc := WALL_LDT();
		// The warning is LOCAL_LDT's own, at its callers.
		{allow 'warn-pragma'}
		LOCAL_LDT := LINT_TO_LDT(LDT_TO_LINT(utc) + LTIME_TO_LINT(LOCAL_OFFSET(IN := utc)));
	END_FUNCTION

	/* A pulse of a fixed length.

	   A rising edge of `IN` sets `Q` for `PT`, whatever `IN` does meanwhile. A new
	   pulse starts on the next rising edge after this one has ended.

	   # Examples

	   ```iecst
	   VAR
	       pulse: TP_TIME;
	   END_VAR

	   pulse(IN := trigger, PT := T#5s);
	   valve := pulse.Q;  // open for five seconds
	   ```
	*/
	{must_call}
	{once}
	FUNCTION_BLOCK TP_TIME
		VAR_INPUT
			IN: BOOL;
			PT: TIME;
		END_VAR
		VAR_OUTPUT
			Q: BOOL := FALSE;
			ET: TIME
		END_VAR
		VAR NON_RETAIN
			STATE: SINT := 0;
			PREV_IN: BOOL := FALSE;
			CURRENT_TIME, START_TIME: TIME;
		END_VAR

		CURRENT_TIME := PLC_TIME();
		IF ((STATE = 0) AND NOT (PREV_IN) AND IN) THEN
			STATE := 1;
			START_TIME := CURRENT_TIME;
		ELSIF ((STATE = 1) AND (CURRENT_TIME - START_TIME >= PT)) THEN
			STATE := 2;
		END_IF;
		IF ((STATE = 2) AND NOT (IN)) THEN
			STATE := 0;
		END_IF;
		IF (STATE = 1) THEN
			ET := CURRENT_TIME - START_TIME;
		ELSIF (STATE = 2) THEN
			ET := PT;
		ELSE
			ET := T#0s;
		END_IF;
		Q := (STATE = 1);
		PREV_IN := IN;
	END_FUNCTION_BLOCK

	TYPE TP: TP_TIME END_TYPE

	/* [Std.Timers.TP_TIME] in `LTIME`. */
	{must_call}
	{once}
	FUNCTION_BLOCK TP_LTIME
		VAR_INPUT
			IN: BOOL;
			PT: LTIME;
		END_VAR
		VAR_OUTPUT
			Q: BOOL := FALSE;
			ET: LTIME
		END_VAR
		VAR NON_RETAIN
			STATE: SINT := 0;
			PREV_IN: BOOL := FALSE;
			CURRENT_TIME, START_TIME: LTIME;
		END_VAR

		CURRENT_TIME := PLC_LTIME();
		IF ((STATE = 0) AND NOT (PREV_IN) AND IN) THEN
			STATE := 1;
			START_TIME := CURRENT_TIME;
		ELSIF ((STATE = 1) AND (CURRENT_TIME - START_TIME >= PT)) THEN
			STATE := 2;
		END_IF;
		IF ((STATE = 2) AND NOT (IN)) THEN
			STATE := 0;
		END_IF;
		IF (STATE = 1) THEN
			ET := CURRENT_TIME - START_TIME;
		ELSIF (STATE = 2) THEN
			ET := PT;
		ELSE
			ET := LTIME#0s;
		END_IF;
		Q := (STATE = 1);
		PREV_IN := IN;
	END_FUNCTION_BLOCK

	/* Delays turning on.

	   `Q` becomes `TRUE` once `IN` has been `TRUE` for `PT`, and `FALSE` as soon
	   as `IN` is. An `IN` that drops before `PT` starts the delay over.

	   # Examples

	   ```iecst
	   VAR
	       delay: TON_TIME;
	   END_VAR

	   delay(IN := start_signal, PT := T#3s);
	   IF delay.Q THEN
	       // start_signal has held for three seconds
	   END_IF;
	   ```
	*/
	{must_call}
	{once}
	FUNCTION_BLOCK TON_TIME
		VAR_INPUT
			IN: BOOL;
			PT: TIME;
		END_VAR
		VAR_OUTPUT
			Q: BOOL := FALSE;
			ET: TIME;
		END_VAR
		VAR NON_RETAIN
			STATE: SINT := 0;
			PREV_IN: BOOL := FALSE;
			CURRENT_TIME, START_TIME: TIME;
		END_VAR

		CURRENT_TIME := PLC_TIME();
		IF (NOT (IN)) THEN
			STATE := 0;
		ELSIF ((STATE = 0) AND NOT (PREV_IN)) THEN
			STATE := 1;
			START_TIME := CURRENT_TIME;
		ELSIF ((STATE = 1) AND (CURRENT_TIME - START_TIME >= PT)) THEN
			STATE := 2;
		END_IF;
		IF (STATE = 1) THEN
			ET := CURRENT_TIME - START_TIME;
		ELSIF (STATE = 2) THEN
			ET := PT;
		ELSE
			ET := T#0s;
		END_IF;
		Q := (STATE = 2);
		PREV_IN := IN;
	END_FUNCTION_BLOCK

	TYPE TON: TON_TIME END_TYPE

	/* [Std.Timers.TON_TIME] in `LTIME`. */
	{must_call}
	{once}
	FUNCTION_BLOCK TON_LTIME
		VAR_INPUT
			IN: BOOL;
			PT: LTIME;
		END_VAR
		VAR_OUTPUT
			Q: BOOL := FALSE;
			ET: LTIME;
		END_VAR
		VAR NON_RETAIN
			STATE: SINT := 0;
			PREV_IN: BOOL := FALSE;
			CURRENT_TIME, START_TIME: LTIME;
		END_VAR

		CURRENT_TIME := PLC_LTIME();
		IF (NOT (IN)) THEN
			STATE := 0;
		ELSIF ((STATE = 0) AND NOT (PREV_IN)) THEN
			STATE := 1;
			START_TIME := CURRENT_TIME;
		ELSIF ((STATE = 1) AND (CURRENT_TIME - START_TIME >= PT)) THEN
			STATE := 2;
		END_IF;
		IF (STATE = 1) THEN
			ET := CURRENT_TIME - START_TIME;
		ELSIF (STATE = 2) THEN
			ET := PT;
		ELSE
			ET := LTIME#0s;
		END_IF;
		Q := (STATE = 2);
		PREV_IN := IN;
	END_FUNCTION_BLOCK

	/* Delays turning off.

	   `Q` is `TRUE` while `IN` is, and stays `TRUE` for `PT` after `IN` drops. An
	   `IN` that comes back before `PT` starts the delay over.

	   # Examples

	   ```iecst
	   VAR
	       off_delay: TOF_TIME;
	   END_VAR

	   off_delay(IN := motor_running, PT := T#10s);
	   cooling_fan := off_delay.Q;  // runs ten seconds after the motor stops
	   ```
	*/
	{must_call}
	{once}
	FUNCTION_BLOCK TOF_TIME
		VAR_INPUT
			IN: BOOL;
			PT: TIME;
		END_VAR
		VAR_OUTPUT
			Q: BOOL := FALSE;
			ET: TIME;
		END_VAR
		VAR NON_RETAIN
			STATE: SINT := 0;
			PREV_IN: BOOL := FALSE;
			CURRENT_TIME, START_TIME: TIME;
		END_VAR

		CURRENT_TIME := PLC_TIME();
		IF (IN) THEN
			STATE := 0;
		ELSIF ((STATE = 0) AND PREV_IN) THEN
			STATE := 1;
			START_TIME := CURRENT_TIME;
		ELSIF ((STATE = 1) AND (CURRENT_TIME - START_TIME >= PT)) THEN
			STATE := 2;
		END_IF;
		IF (STATE = 1) THEN
			ET := CURRENT_TIME - START_TIME;
		ELSIF (STATE = 2) THEN
			ET := PT;
		ELSE
			ET := T#0s;
		END_IF;
		Q := IN OR (STATE = 1);
		PREV_IN := IN;
	END_FUNCTION_BLOCK

	TYPE TOF: TOF_TIME END_TYPE

	/* [Std.Timers.TOF_TIME] in `LTIME`. */
	{must_call}
	{once}
	FUNCTION_BLOCK TOF_LTIME
		VAR_INPUT
			IN: BOOL;
			PT: LTIME;
		END_VAR
		VAR_OUTPUT
			Q: BOOL := FALSE;
			ET: LTIME;
		END_VAR
		VAR NON_RETAIN
			STATE: SINT := 0;
			PREV_IN: BOOL := FALSE;
			CURRENT_TIME, START_TIME: LTIME;
		END_VAR

		CURRENT_TIME := PLC_LTIME();
		IF (IN) THEN
			STATE := 0;
		ELSIF ((STATE = 0) AND PREV_IN) THEN
			STATE := 1;
			START_TIME := CURRENT_TIME;
		ELSIF ((STATE = 1) AND (CURRENT_TIME - START_TIME >= PT)) THEN
			STATE := 2;
		END_IF;
		IF (STATE = 1) THEN
			ET := CURRENT_TIME - START_TIME;
		ELSIF (STATE = 2) THEN
			ET := PT;
		ELSE
			ET := LTIME#0s;
		END_IF;
		Q := IN OR (STATE = 1);
		PREV_IN := IN;
	END_FUNCTION_BLOCK

	NAMESPACE Test
		USING Std.Unit;
		USING Std.Timers;

		// A test that waits for the clock is a block: it calls each timer once
		// per cycle, as a program does, and is DONE in the cycle where what it
		// waits for has happened.

		// -- TON (On-Delay Timer) ------------------------------------

		{test}
		FUNCTION_BLOCK test_ton_expires
			VAR_OUTPUT
				DONE: BOOL;
			END_VAR
			VAR
				timer: TON_TIME;
			END_VAR
			timer(IN := TRUE, PT := T#1ms);
			DONE := timer.Q;
		END_FUNCTION_BLOCK

		{test}
		FUNCTION test_ton_not_started
			VAR
				timer: TON_TIME;
			END_VAR
			timer(IN := FALSE, PT := T#1ms);
			ASSERT(NOT timer.Q, 'TON Q should be FALSE when IN is FALSE');
		END_FUNCTION

		{test}
		FUNCTION test_ton_reset
			VAR
				timer: TON_TIME;
			END_VAR
			timer(IN := TRUE, PT := T#100ms);
			ASSERT(NOT timer.Q, 'TON Q should be FALSE immediately');
			timer(IN := FALSE, PT := T#100ms);
			ASSERT(NOT timer.Q, 'TON Q should be FALSE after reset');
			ASSERT(timer.ET = T#0s, 'TON ET should be 0 after reset');
		END_FUNCTION

		// -- TOF (Off-Delay Timer) -----------------------------------

		{test}
		FUNCTION test_tof_stays_true_after_falling_edge
			VAR
				timer: TOF_TIME;
			END_VAR
			// Rising edge: Q becomes TRUE immediately
			timer(IN := TRUE, PT := T#100ms);
			ASSERT(timer.Q, 'TOF Q should be TRUE when IN is TRUE');
			// Falling edge: Q stays TRUE during delay
			timer(IN := FALSE, PT := T#100ms);
			ASSERT(timer.Q, 'TOF Q should stay TRUE during off-delay');
		END_FUNCTION

		{test}
		FUNCTION_BLOCK test_tof_expires
			VAR_OUTPUT
				DONE: BOOL;
			END_VAR
			VAR
				timer: TOF_TIME;
				step: INT;
			END_VAR
			// IN on the first cycle, off from the second.
			timer(IN := step = 0, PT := T#1ms);
			IF step = 0 THEN
				step := 1;
			ELSE
				DONE := NOT timer.Q;
			END_IF;
		END_FUNCTION_BLOCK

		{test}
		FUNCTION test_tof_reset_on_rising_edge
			VAR
				timer: TOF_TIME;
			END_VAR
			timer(IN := TRUE, PT := T#1ms);
			timer(IN := FALSE, PT := T#1ms);
			// Re-assert IN before timer expires
			timer(IN := TRUE, PT := T#1ms);
			ASSERT(timer.Q, 'TOF Q should be TRUE after re-assertion');
		END_FUNCTION

		// -- TP (Pulse Timer) ----------------------------------------

		{test}
		FUNCTION test_tp_pulse_starts
			VAR
				timer: TP_TIME;
			END_VAR
			timer(IN := TRUE, PT := T#100ms);
			ASSERT(timer.Q, 'TP Q should be TRUE on rising edge');
		END_FUNCTION

		{test}
		FUNCTION_BLOCK test_tp_pulse_expires
			VAR_OUTPUT
				DONE: BOOL;
			END_VAR
			VAR
				timer: TP_TIME;
			END_VAR
			timer(IN := TRUE, PT := T#1ms);
			DONE := NOT timer.Q;
		END_FUNCTION_BLOCK

		{test}
		FUNCTION test_tp_ignores_input_during_pulse
			VAR
				timer: TP_TIME;
			END_VAR
			timer(IN := TRUE, PT := T#100ms);
			ASSERT(timer.Q, 'TP Q should be TRUE');
			// Dropping IN during pulse doesn't affect Q
			timer(IN := FALSE, PT := T#100ms);
			ASSERT(timer.Q, 'TP Q should stay TRUE during pulse even if IN drops');
		END_FUNCTION

		// --- TON must NOT fire before PT: an instant-expiry TON (PT ignored
		// or inverted compare) passes every test above that waits for Q ---

		{test}
		FUNCTION test_ton_stays_false_before_expiry
			VAR
				timer: TON_TIME;
				i: INT;
			END_VAR
			timer(IN := TRUE, PT := T#1h);
			FOR i := 1 TO 10 DO
				timer(IN := TRUE, PT := T#1h);
				ASSERT(NOT timer.Q, 'TON must not fire long before PT elapses');
			END_FOR;
			ASSERT(timer.ET < T#1h, 'ET tracks elapsed time below PT');
		END_FUNCTION

		{test}
		FUNCTION_BLOCK test_ton_et_clamps_at_pt
			VAR_OUTPUT
				DONE: BOOL;
			END_VAR
			VAR
				timer: TON_TIME;
				step: INT;
				t0: TIME;
			END_VAR
			timer(IN := TRUE, PT := T#1ms);
			IF step = 0 AND timer.Q THEN
				t0 := PLC_TIME();
				step := 1;
			END_IF;
			IF step = 1 THEN
				// IN held 2 ms past the deadline: ET stays at PT.
				ASSERT(timer.Q AND timer.ET = T#1ms, 'ET is exactly PT after expiry');
				DONE := PLC_TIME() - t0 >= T#2ms;
			END_IF;
		END_FUNCTION_BLOCK

		// --- TP terminal state: no auto-refire while IN is held, and a fresh
		// rising edge after release starts a new pulse ---

		{test}
		FUNCTION_BLOCK test_tp_post_pulse_retrigger
			VAR_OUTPUT
				DONE: BOOL;
			END_VAR
			VAR
				timer: TP_TIME;
				step: INT;
				t0: TIME;
			END_VAR
			// IN held, released for the one cycle of step 2, then held again.
			timer(IN := step <> 2, PT := T#1ms);
			IF step = 0 AND NOT timer.Q THEN
				// The pulse has ended.
				t0 := PLC_TIME();
				step := 1;
			END_IF;
			IF step = 1 THEN
				// IN held 2 ms past the pulse: ET stays at PT, and no new pulse.
				ASSERT(timer.ET = T#1ms, 'ET clamps at PT when the pulse ends');
				ASSERT(NOT timer.Q, 'held-high IN must not refire the pulse');
				IF PLC_TIME() - t0 >= T#2ms THEN
					step := 2;
				END_IF;
			ELSIF step = 2 THEN
				step := 3;
			ELSIF step = 3 THEN
				ASSERT(timer.Q, 'a new rising edge after release starts a new pulse');
				DONE := TRUE;
			END_IF;
		END_FUNCTION_BLOCK

		// --- TOF: re-asserting IN cancels the pending expiry; the NEXT
		// falling edge must get a fresh deadline, not the stale one ---

		{test}
		FUNCTION_BLOCK test_tof_fresh_deadline_after_reassert
			VAR_OUTPUT
				DONE: BOOL;
			END_VAR
			VAR
				timer: TOF_TIME;
				step: INT;
				t0, t1: TIME;
			END_VAR
			// IN rises, falls, rises again until the first off-delay's deadline
			// has passed, then falls for good.
			timer(IN := step = 0 OR step = 2, PT := T#50ms);
			IF step = 0 THEN
				step := 1;
			ELSIF step = 1 THEN
				// The first off-delay started in this cycle.
				t0 := PLC_TIME();
				step := 2;
			ELSIF step = 2 THEN
				IF PLC_TIME() - t0 >= T#60ms THEN
					// IN falls in the next cycle, after t1.
					t1 := PLC_TIME();
					step := 3;
				END_IF;
			ELSIF step = 3 THEN
				// New falling edge: deadline must be now+PT, not the stale t0+PT.
				ASSERT(timer.Q, 'TOF must use a fresh deadline for a new falling edge');
				step := 4;
			ELSIF NOT timer.Q THEN
				ASSERT(PLC_TIME() - t1 >= T#50ms, 'TOF must hold Q for PT after the new falling edge');
				DONE := TRUE;
			END_IF;
		END_FUNCTION_BLOCK

		{test}
		FUNCTION_BLOCK test_tof_et_clamps_at_pt
			VAR_OUTPUT
				DONE: BOOL;
			END_VAR
			VAR
				timer: TOF_TIME;
				step: INT;
				t0: TIME;
			END_VAR
			// IN on the first cycle, off from the second.
			timer(IN := step = 0, PT := T#1ms);
			IF step = 0 THEN
				step := 1;
			ELSIF step = 1 AND NOT timer.Q THEN
				t0 := PLC_TIME();
				step := 2;
			END_IF;
			IF step = 2 THEN
				// IN off 2 ms past the deadline: ET stays at PT.
				ASSERT(NOT timer.Q AND timer.ET = T#1ms, 'ET is exactly PT after the off-delay expires');
				DONE := PLC_TIME() - t0 >= T#2ms;
			END_IF;
		END_FUNCTION_BLOCK

		// --- PT = 0 (pins current behavior: the deadline check runs on the
		// call AFTER the starting edge, so a zero preset needs two calls) ---

		{test}
		FUNCTION test_pt_zero_pins_current_behavior
			VAR
				ton_timer: TON_TIME;
				tp_timer: TP_TIME;
			END_VAR
			ton_timer(IN := TRUE, PT := T#0s);
			ASSERT(NOT ton_timer.Q, 'TON PT=0: edge call does not evaluate the deadline yet');
			ton_timer(IN := TRUE, PT := T#0s);
			ASSERT(ton_timer.Q, 'TON PT=0: fires on the next call');
			tp_timer(IN := TRUE, PT := T#0s);
			ASSERT(tp_timer.Q, 'TP PT=0: pulse starts on the edge call');
			tp_timer(IN := TRUE, PT := T#0s);
			ASSERT(NOT tp_timer.Q, 'TP PT=0: pulse over on the next call');
		END_FUNCTION

		// -- the LTIME variants run the same machine on the ns clock --

		{test}
		FUNCTION_BLOCK test_ton_ltime_expires
			VAR_OUTPUT
				DONE: BOOL;
			END_VAR
			VAR
				timer: TON_LTIME;
			END_VAR
			timer(IN := TRUE, PT := LTIME#1ms);
			IF timer.Q THEN
				ASSERT(timer.ET = LTIME#1ms, 'TON_LTIME ET is exactly PT after expiry');
				DONE := TRUE;
			END_IF;
		END_FUNCTION_BLOCK

		{test}
		FUNCTION_BLOCK test_tof_ltime_expires
			VAR_OUTPUT
				DONE: BOOL;
			END_VAR
			VAR
				timer: TOF_LTIME;
				step: INT;
			END_VAR
			// IN on the first cycle, off from the second.
			timer(IN := step = 0, PT := LTIME#1ms);
			IF step = 0 THEN
				ASSERT(timer.Q, 'TOF_LTIME Q should be TRUE while IN is TRUE');
				step := 1;
			ELSIF NOT timer.Q THEN
				ASSERT(timer.ET = LTIME#1ms, 'TOF_LTIME ET clamps at PT after expiry');
				DONE := TRUE;
			END_IF;
		END_FUNCTION_BLOCK

		{test}
		FUNCTION_BLOCK test_tp_ltime_pulse
			VAR_OUTPUT
				DONE: BOOL;
			END_VAR
			VAR
				timer: TP_LTIME;
				step: INT;
			END_VAR
			timer(IN := TRUE, PT := LTIME#1ms);
			IF step = 0 THEN
				ASSERT(timer.Q, 'TP_LTIME Q should be TRUE on rising edge');
				step := 1;
			ELSIF NOT timer.Q THEN
				ASSERT(timer.ET = LTIME#1ms, 'TP_LTIME ET clamps at PT when the pulse ends');
				DONE := TRUE;
			END_IF;
		END_FUNCTION_BLOCK

		// -- the standard names are aliases; instances declared through
		// them must build, call, and expose the outputs --

		{test}
		FUNCTION_BLOCK test_standard_names_are_usable
			VAR_OUTPUT
				DONE: BOOL;
			END_VAR
			VAR
				pulse: TP;
				on_delay: TON;
				off_delay: TOF;
				step: INT;
			END_VAR
			pulse(IN := TRUE, PT := T#100ms);
			on_delay(IN := TRUE, PT := T#1ms);
			// IN on the first cycle, off from the second.
			off_delay(IN := step = 0, PT := T#100ms);
			IF step = 0 THEN
				ASSERT(pulse.Q, 'a TP-typed instance pulses on the rising edge');
				step := 1;
			ELSIF step = 1 THEN
				ASSERT(off_delay.Q, 'a TOF-typed instance holds Q through the off-delay');
				step := 2;
			ELSIF on_delay.Q THEN
				ASSERT(on_delay.ET = T#1ms, 'a TON-typed instance expires at PT');
				DONE := TRUE;
			END_IF;
		END_FUNCTION_BLOCK

		// --- the clock itself ---

		{test}
		FUNCTION test_plc_time_monotonic
			VAR
				t1, t2: TIME;
			END_VAR
			t1 := PLC_TIME();
			t2 := PLC_TIME();
			// TIME wraps every 49.7 days: compare the difference, as a timer does.
			ASSERT(t2 - t1 >= T#0s, 'PLC_TIME must be monotonic');
		END_FUNCTION

		{test}
		FUNCTION test_plc_ltime_monotonic
			VAR
				t1, t2: LTIME;
			END_VAR
			t1 := PLC_LTIME();
			t2 := PLC_LTIME();
			ASSERT(t2 - t1 >= LTIME#0s, 'PLC_LTIME must be monotonic');
		END_FUNCTION

		// -- The wall clock ------------------------------------------

		{test}
		FUNCTION test_wall_clock_is_after_2026
			ASSERT(WALL_LDT() > LDT#2026-01-01-00:00:00, 'WALL_LDT is before 2026');
			ASSERT(WALL_DT() > DT#2026-01-01-00:00:00, 'WALL_DT is before 2026');
		END_FUNCTION

		{test}
		{allow 'warn-pragma'}
		FUNCTION test_local_clock_is_the_wall_clock_shifted
			VAR
				wall, local : LDT;
				offset : LTIME;
				shift : LINT;
			END_VAR
			wall := WALL_LDT();
			offset := LOCAL_OFFSET(IN := wall);
			local := LOCAL_LDT();
			ASSERT(offset >= LT#-18h AND offset <= LT#18h, 'the zone is more than a day from UTC');
			// `local` was read after `wall`: the readings are a moment apart.
			shift := LDT_TO_LINT(local) - LDT_TO_LINT(wall) - LTIME_TO_LINT(offset);
			ASSERT(shift >= LINT#0 AND shift < LINT#1000000000, 'LOCAL_LDT is not WALL_LDT shifted by LOCAL_OFFSET');
		END_FUNCTION
	END_NAMESPACE
END_NAMESPACE

(* ---- Unit.st ---- *)
/*
Assertions for `{test}` functions.

A failed assertion raises, and `rk test` reports the test as failed with
its message.
*/
NAMESPACE Std.Unit
	USING Std.Strings;

	/* Raises `message` when `value` is `FALSE`.

	   # Examples

	   ```iecst
	   ASSERT(level < 100, 'the tank overflowed');
	   ```
	*/
	FUNCTION ASSERT
		VAR_INPUT
			value: BOOL;
			message: STRING := '';
		END_VAR

		IF NOT value THEN
			__RAISE(CONCAT('assertion failed: ', message));
		END_IF
	END_FUNCTION

	/* Raises `message` when `value` and `target` differ.

	   There is one overload per elementary type. Both must have the same type,
	   so write a typed literal where the compiler cannot tell: `INT#5`.

	   # Examples

	   ```iecst
	   ASSERT_EQ(ABS(-5), 5, 'ABS of a negative');
	   ```
	*/
	FUNCTION ASSERT_EQ
		VAR_INPUT
			value: BOOL;
			target: BOOL;
			message: STRING := '';
		END_VAR

		IF value <> target THEN
			__RAISE(CONCAT('assertion failed: ', message));
		END_IF
	END_FUNCTION

	FUNCTION ASSERT_EQ
		VAR_INPUT
			value: SINT;
			target: SINT;
			message: STRING := '';
		END_VAR

		IF value <> target THEN
			__RAISE(CONCAT('assertion failed: ', message));
		END_IF
	END_FUNCTION

	FUNCTION ASSERT_EQ
		VAR_INPUT
			value: INT;
			target: INT;
			message: STRING := '';
		END_VAR

		IF value <> target THEN
			__RAISE(CONCAT('assertion failed: ', message));
		END_IF
	END_FUNCTION

	FUNCTION ASSERT_EQ
		VAR_INPUT
			value: DINT;
			target: DINT;
			message: STRING := '';
		END_VAR

		IF value <> target THEN
			__RAISE(CONCAT('assertion failed: ', message));
		END_IF
	END_FUNCTION

	FUNCTION ASSERT_EQ
		VAR_INPUT
			value: LINT;
			target: LINT;
			message: STRING := '';
		END_VAR

		IF value <> target THEN
			__RAISE(CONCAT('assertion failed: ', message));
		END_IF
	END_FUNCTION

	FUNCTION ASSERT_EQ
		VAR_INPUT
			value: USINT;
			target: USINT;
			message: STRING := '';
		END_VAR

		IF value <> target THEN
			__RAISE(CONCAT('assertion failed: ', message));
		END_IF
	END_FUNCTION

	FUNCTION ASSERT_EQ
		VAR_INPUT
			value: UINT;
			target: UINT;
			message: STRING := '';
		END_VAR

		IF value <> target THEN
			__RAISE(CONCAT('assertion failed: ', message));
		END_IF
	END_FUNCTION

	FUNCTION ASSERT_EQ
		VAR_INPUT
			value: UDINT;
			target: UDINT;
			message: STRING := '';
		END_VAR

		IF value <> target THEN
			__RAISE(CONCAT('assertion failed: ', message));
		END_IF
	END_FUNCTION

	FUNCTION ASSERT_EQ
		VAR_INPUT
			value: ULINT;
			target: ULINT;
			message: STRING := '';
		END_VAR

		IF value <> target THEN
			__RAISE(CONCAT('assertion failed: ', message));
		END_IF
	END_FUNCTION

	FUNCTION ASSERT_EQ
		VAR_INPUT
			value: BYTE;
			target: BYTE;
			message: STRING := '';
		END_VAR

		IF value <> target THEN
			__RAISE(CONCAT('assertion failed: ', message));
		END_IF
	END_FUNCTION

	FUNCTION ASSERT_EQ
		VAR_INPUT
			value: WORD;
			target: WORD;
			message: STRING := '';
		END_VAR

		IF value <> target THEN
			__RAISE(CONCAT('assertion failed: ', message));
		END_IF
	END_FUNCTION

	FUNCTION ASSERT_EQ
		VAR_INPUT
			value: DWORD;
			target: DWORD;
			message: STRING := '';
		END_VAR

		IF value <> target THEN
			__RAISE(CONCAT('assertion failed: ', message));
		END_IF
	END_FUNCTION

	FUNCTION ASSERT_EQ
		VAR_INPUT
			value: LWORD;
			target: LWORD;
			message: STRING := '';
		END_VAR

		IF value <> target THEN
			__RAISE(CONCAT('assertion failed: ', message));
		END_IF
	END_FUNCTION

	// Equal means the same value, not one within a tolerance.
	{allow 'float-equality'}
	FUNCTION ASSERT_EQ
		VAR_INPUT
			value: REAL;
			target: REAL;
			message: STRING := '';
		END_VAR

		IF value <> target THEN
			__RAISE(CONCAT('assertion failed: ', message));
		END_IF
	END_FUNCTION

	// Equal means the same value, not one within a tolerance.
	{allow 'float-equality'}
	FUNCTION ASSERT_EQ
		VAR_INPUT
			value: LREAL;
			target: LREAL;
			message: STRING := '';
		END_VAR

		IF value <> target THEN
			__RAISE(CONCAT('assertion failed: ', message));
		END_IF
	END_FUNCTION

	FUNCTION ASSERT_EQ
		VAR_INPUT
			value: TIME;
			target: TIME;
			message: STRING := '';
		END_VAR

		IF value <> target THEN
			__RAISE(CONCAT('assertion failed: ', message));
		END_IF
	END_FUNCTION

	FUNCTION ASSERT_EQ
		VAR_INPUT
			value: LTIME;
			target: LTIME;
			message: STRING := '';
		END_VAR

		IF value <> target THEN
			__RAISE(CONCAT('assertion failed: ', message));
		END_IF
	END_FUNCTION

	FUNCTION ASSERT_EQ
		VAR_INPUT
			value: STRING[255];
			target: STRING[255];
			message: STRING := '';
		END_VAR

		IF value <> target THEN
			__RAISE(CONCAT('assertion failed: ', message));
		END_IF
	END_FUNCTION

	FUNCTION ASSERT_EQ
		VAR_INPUT
			value: CHAR;
			target: CHAR;
			message: STRING := '';
		END_VAR

		IF value <> target THEN
			__RAISE(CONCAT('assertion failed: ', message));
		END_IF
	END_FUNCTION

	/* Raises `message` when `value` and `target` are equal.

	   There is one overload per elementary type.
	*/
	FUNCTION ASSERT_NEQ
		VAR_INPUT
			value: BOOL;
			target: BOOL;
			message: STRING := '';
		END_VAR

		IF value = target THEN
			__RAISE(CONCAT('assertion failed: ', message));
		END_IF
	END_FUNCTION

	FUNCTION ASSERT_NEQ
		VAR_INPUT
			value: SINT;
			target: SINT;
			message: STRING := '';
		END_VAR

		IF value = target THEN
			__RAISE(CONCAT('assertion failed: ', message));
		END_IF
	END_FUNCTION

	FUNCTION ASSERT_NEQ
		VAR_INPUT
			value: INT;
			target: INT;
			message: STRING := '';
		END_VAR

		IF value = target THEN
			__RAISE(CONCAT('assertion failed: ', message));
		END_IF
	END_FUNCTION

	FUNCTION ASSERT_NEQ
		VAR_INPUT
			value: DINT;
			target: DINT;
			message: STRING := '';
		END_VAR

		IF value = target THEN
			__RAISE(CONCAT('assertion failed: ', message));
		END_IF
	END_FUNCTION

	FUNCTION ASSERT_NEQ
		VAR_INPUT
			value: LINT;
			target: LINT;
			message: STRING := '';
		END_VAR

		IF value = target THEN
			__RAISE(CONCAT('assertion failed: ', message));
		END_IF
	END_FUNCTION

	FUNCTION ASSERT_NEQ
		VAR_INPUT
			value: USINT;
			target: USINT;
			message: STRING := '';
		END_VAR

		IF value = target THEN
			__RAISE(CONCAT('assertion failed: ', message));
		END_IF
	END_FUNCTION

	FUNCTION ASSERT_NEQ
		VAR_INPUT
			value: UINT;
			target: UINT;
			message: STRING := '';
		END_VAR

		IF value = target THEN
			__RAISE(CONCAT('assertion failed: ', message));
		END_IF
	END_FUNCTION

	FUNCTION ASSERT_NEQ
		VAR_INPUT
			value: UDINT;
			target: UDINT;
			message: STRING := '';
		END_VAR

		IF value = target THEN
			__RAISE(CONCAT('assertion failed: ', message));
		END_IF
	END_FUNCTION

	FUNCTION ASSERT_NEQ
		VAR_INPUT
			value: ULINT;
			target: ULINT;
			message: STRING := '';
		END_VAR

		IF value = target THEN
			__RAISE(CONCAT('assertion failed: ', message));
		END_IF
	END_FUNCTION

	FUNCTION ASSERT_NEQ
		VAR_INPUT
			value: BYTE;
			target: BYTE;
			message: STRING := '';
		END_VAR

		IF value = target THEN
			__RAISE(CONCAT('assertion failed: ', message));
		END_IF
	END_FUNCTION

	FUNCTION ASSERT_NEQ
		VAR_INPUT
			value: WORD;
			target: WORD;
			message: STRING := '';
		END_VAR

		IF value = target THEN
			__RAISE(CONCAT('assertion failed: ', message));
		END_IF
	END_FUNCTION

	FUNCTION ASSERT_NEQ
		VAR_INPUT
			value: DWORD;
			target: DWORD;
			message: STRING := '';
		END_VAR

		IF value = target THEN
			__RAISE(CONCAT('assertion failed: ', message));
		END_IF
	END_FUNCTION

	FUNCTION ASSERT_NEQ
		VAR_INPUT
			value: LWORD;
			target: LWORD;
			message: STRING := '';
		END_VAR

		IF value = target THEN
			__RAISE(CONCAT('assertion failed: ', message));
		END_IF
	END_FUNCTION

	// Equal means the same value, not one within a tolerance.
	{allow 'float-equality'}
	FUNCTION ASSERT_NEQ
		VAR_INPUT
			value: REAL;
			target: REAL;
			message: STRING := '';
		END_VAR

		IF value = target THEN
			__RAISE(CONCAT('assertion failed: ', message));
		END_IF
	END_FUNCTION

	// Equal means the same value, not one within a tolerance.
	{allow 'float-equality'}
	FUNCTION ASSERT_NEQ
		VAR_INPUT
			value: LREAL;
			target: LREAL;
			message: STRING := '';
		END_VAR

		IF value = target THEN
			__RAISE(CONCAT('assertion failed: ', message));
		END_IF
	END_FUNCTION

	FUNCTION ASSERT_NEQ
		VAR_INPUT
			value: TIME;
			target: TIME;
			message: STRING := '';
		END_VAR

		IF value = target THEN
			__RAISE(CONCAT('assertion failed: ', message));
		END_IF
	END_FUNCTION

	FUNCTION ASSERT_NEQ
		VAR_INPUT
			value: LTIME;
			target: LTIME;
			message: STRING := '';
		END_VAR

		IF value = target THEN
			__RAISE(CONCAT('assertion failed: ', message));
		END_IF
	END_FUNCTION

	FUNCTION ASSERT_NEQ
		VAR_INPUT
			value: STRING[255];
			target: STRING[255];
			message: STRING := '';
		END_VAR

		IF value = target THEN
			__RAISE(CONCAT('assertion failed: ', message));
		END_IF
	END_FUNCTION

	FUNCTION ASSERT_NEQ
		VAR_INPUT
			value: CHAR;
			target: CHAR;
			message: STRING := '';
		END_VAR

		IF value = target THEN
			__RAISE(CONCAT('assertion failed: ', message));
		END_IF
	END_FUNCTION

	// The six calendar types

	FUNCTION ASSERT_EQ
		VAR_INPUT
			value: DATE;
			target: DATE;
			message: STRING := '';
		END_VAR

		IF value <> target THEN
			__RAISE(CONCAT('assertion failed: ', message));
		END_IF
	END_FUNCTION

	FUNCTION ASSERT_EQ
		VAR_INPUT
			value: LDATE;
			target: LDATE;
			message: STRING := '';
		END_VAR

		IF value <> target THEN
			__RAISE(CONCAT('assertion failed: ', message));
		END_IF
	END_FUNCTION

	FUNCTION ASSERT_EQ
		VAR_INPUT
			value: TIME_OF_DAY;
			target: TIME_OF_DAY;
			message: STRING := '';
		END_VAR

		IF value <> target THEN
			__RAISE(CONCAT('assertion failed: ', message));
		END_IF
	END_FUNCTION

	FUNCTION ASSERT_EQ
		VAR_INPUT
			value: LTIME_OF_DAY;
			target: LTIME_OF_DAY;
			message: STRING := '';
		END_VAR

		IF value <> target THEN
			__RAISE(CONCAT('assertion failed: ', message));
		END_IF
	END_FUNCTION

	FUNCTION ASSERT_EQ
		VAR_INPUT
			value: DATE_AND_TIME;
			target: DATE_AND_TIME;
			message: STRING := '';
		END_VAR

		IF value <> target THEN
			__RAISE(CONCAT('assertion failed: ', message));
		END_IF
	END_FUNCTION

	FUNCTION ASSERT_EQ
		VAR_INPUT
			value: LDATE_AND_TIME;
			target: LDATE_AND_TIME;
			message: STRING := '';
		END_VAR

		IF value <> target THEN
			__RAISE(CONCAT('assertion failed: ', message));
		END_IF
	END_FUNCTION

	FUNCTION ASSERT_NEQ
		VAR_INPUT
			value: DATE;
			target: DATE;
			message: STRING := '';
		END_VAR

		IF value = target THEN
			__RAISE(CONCAT('assertion failed: ', message));
		END_IF
	END_FUNCTION

	FUNCTION ASSERT_NEQ
		VAR_INPUT
			value: LDATE;
			target: LDATE;
			message: STRING := '';
		END_VAR

		IF value = target THEN
			__RAISE(CONCAT('assertion failed: ', message));
		END_IF
	END_FUNCTION

	FUNCTION ASSERT_NEQ
		VAR_INPUT
			value: TIME_OF_DAY;
			target: TIME_OF_DAY;
			message: STRING := '';
		END_VAR

		IF value = target THEN
			__RAISE(CONCAT('assertion failed: ', message));
		END_IF
	END_FUNCTION

	FUNCTION ASSERT_NEQ
		VAR_INPUT
			value: LTIME_OF_DAY;
			target: LTIME_OF_DAY;
			message: STRING := '';
		END_VAR

		IF value = target THEN
			__RAISE(CONCAT('assertion failed: ', message));
		END_IF
	END_FUNCTION

	FUNCTION ASSERT_NEQ
		VAR_INPUT
			value: DATE_AND_TIME;
			target: DATE_AND_TIME;
			message: STRING := '';
		END_VAR

		IF value = target THEN
			__RAISE(CONCAT('assertion failed: ', message));
		END_IF
	END_FUNCTION

	FUNCTION ASSERT_NEQ
		VAR_INPUT
			value: LDATE_AND_TIME;
			target: LDATE_AND_TIME;
			message: STRING := '';
		END_VAR

		IF value = target THEN
			__RAISE(CONCAT('assertion failed: ', message));
		END_IF
	END_FUNCTION

	NAMESPACE Test
		USING Std.Unit;

		{test}
		FUNCTION test_assert_eq_accepts_every_date_and_time_type
			ASSERT_EQ(value := D#2024-02-29, target := D#2024-02-29, message := 'DATE');
			ASSERT_EQ(value := LD#2024-02-29, target := LD#2024-02-29, message := 'LDATE');
			ASSERT_EQ(value := TOD#12:30:45.123, target := TOD#12:30:45.123, message := 'TOD');
			ASSERT_EQ(value := LTOD#12:30:45.123456789, target := LTOD#12:30:45.123456789, message := 'LTOD');
			ASSERT_EQ(value := DT#2024-02-29-12:30:45, target := DT#2024-02-29-12:30:45, message := 'DT');
			ASSERT_EQ(value := LDT#2024-02-29-12:30:45.5, target := LDT#2024-02-29-12:30:45.5, message := 'LDT');
		END_FUNCTION

		{test}
		FUNCTION test_assert_neq_sees_a_different_date_or_time
			ASSERT_NEQ(value := D#2024-02-29, target := D#2024-03-01, message := 'DATE');
			ASSERT_NEQ(value := LD#1969-12-31, target := LD#1970-01-01, message := 'LDATE, across the epoch');
			ASSERT_NEQ(value := TOD#12:30:45, target := TOD#12:30:45.001, message := 'TOD, a millisecond apart');
			ASSERT_NEQ(value := LTOD#12:30:45, target := LTOD#12:30:45.000000001, message := 'LTOD, a nanosecond apart');
			ASSERT_NEQ(value := DT#2024-02-29-12:30:45, target := DT#2024-02-29-12:30:46, message := 'DT');
			ASSERT_NEQ(value := LDT#2024-02-29-12:30:45.5, target := LDT#2024-02-29-12:30:45.6, message := 'LDT');
		END_FUNCTION
	END_NAMESPACE

END_NAMESPACE

(* ---- Bistable.st ---- *)
/*
Latches and a semaphore.

[Std.Bistable.SR] and [Std.Bistable.RS] differ only in which input wins
when both are `TRUE`.
*/
NAMESPACE Std.Bistable

	/* A latch where set wins.

	   `S1` sets `Q1` and `R` resets it. `Q1` keeps its value when both are
	   `FALSE`, and is set when both are `TRUE`.

	   # Examples

	   ```iecst
	   VAR
	       latch: SR;
	   END_VAR

	   latch(start_btn, stop_btn);
	   motor := latch.Q1;
	   ```
	*/
	{must_call}
	{once}
	FUNCTION_BLOCK SR
		VAR_INPUT
			S1, R: BOOL;
		END_VAR
		VAR_OUTPUT
			Q1: BOOL;
		END_VAR Q1 := S1 OR ((NOT R) AND Q1);
	END_FUNCTION_BLOCK

	/* A latch where reset wins.

	   `S` sets `Q1` and `R1` resets it. `Q1` keeps its value when both are
	   `FALSE`, and is reset when both are `TRUE`.

	   # Examples

	   ```iecst
	   VAR
	       latch: RS;
	   END_VAR

	   latch(start_btn, emergency_stop);
	   motor := latch.Q1;
	   ```
	*/
	{must_call}
	{once}
	FUNCTION_BLOCK RS
		VAR_INPUT
			S, R1: BOOL;
		END_VAR
		VAR_OUTPUT
			Q1: BOOL;
		END_VAR Q1 := (NOT R1) AND (S OR Q1);
	END_FUNCTION_BLOCK

	/* A semaphore over a shared resource.

	   `CLAIM` takes it and `RELEASE` frees it. `BUSY` is `TRUE` when the call
	   claimed a semaphore that was already taken, so a caller owns the resource
	   when it claims and `BUSY` is `FALSE`. A claim wins over a release made in
	   the same call.

	   # Examples

	   ```iecst
	   VAR
	       sem: SEMA;
	   END_VAR

	   sem(CLAIM := want_it, RELEASE := done_with_it);
	   IF NOT sem.BUSY THEN
	       // the resource is ours
	   END_IF;
	   ```
	*/
	{must_call}
	{once}
	FUNCTION_BLOCK SEMA
		VAR_INPUT
			CLAIM, RELEASE: BOOL;
		END_VAR
		VAR_OUTPUT
			BUSY: BOOL;
		END_VAR
		VAR
			X: BOOL;
		END_VAR

		BUSY := X;
		IF CLAIM THEN
			X := TRUE;
		ELSIF RELEASE THEN
			BUSY := FALSE;
			X := FALSE;
		END_IF;
	END_FUNCTION_BLOCK

	NAMESPACE Test
		USING Std.Unit

		{test}
		FUNCTION test_sr_set
			VAR
				latch: SR;
			END_VAR
			latch(TRUE, FALSE);
			ASSERT(latch.Q1);
		END_FUNCTION

		{test}
		FUNCTION test_sr_reset
			VAR
				latch: SR;
			END_VAR
			// First set
			latch(TRUE, FALSE);
			// Then reset
			latch(FALSE, TRUE);
			ASSERT(NOT latch.Q1);
		END_FUNCTION

		{test}
		FUNCTION test_sr_set_dominant
			VAR
				latch: SR;
			END_VAR
			// Both inputs TRUE: set wins
			latch(TRUE, TRUE);
			ASSERT(latch.Q1);
		END_FUNCTION

		{test}
		FUNCTION test_rs_set
			VAR
				latch: RS;
			END_VAR
			latch(TRUE, FALSE);
			ASSERT(latch.Q1);
		END_FUNCTION

		{test}
		FUNCTION test_rs_reset_dominant
			VAR
				latch: RS;
			END_VAR
			// Both inputs TRUE: reset wins
			latch(TRUE, TRUE);
			ASSERT(NOT latch.Q1);
		END_FUNCTION

		// --- the latch must LATCH: state persists through (FALSE, FALSE).
		// A memoryless body (`Q1 := S1`) passes every test above ---

		{test}
		FUNCTION test_sr_holds_state_after_release
			VAR
				latch: SR;
			END_VAR
			latch(TRUE, FALSE);
			latch(FALSE, FALSE);
			ASSERT(latch.Q1, 'SR must stay set once S1 is released');
			latch(FALSE, FALSE);
			ASSERT(latch.Q1, 'and stay set across further idle calls');
		END_FUNCTION

		{test}
		FUNCTION test_sr_stays_reset_after_release
			VAR
				latch: SR;
			END_VAR
			latch(TRUE, FALSE);
			latch(FALSE, TRUE);
			latch(FALSE, FALSE);
			ASSERT(NOT latch.Q1, 'SR must stay reset once R is released');
		END_FUNCTION

		{test}
		FUNCTION test_rs_holds_state_after_release
			VAR
				latch: RS;
			END_VAR
			latch(TRUE, FALSE);
			latch(FALSE, FALSE);
			ASSERT(latch.Q1, 'RS must stay set once S is released');
		END_FUNCTION

		{test}
		FUNCTION test_rs_dominance_is_not_sticky
			VAR
				latch: RS;
			END_VAR
			// Reset-dominant call, then a plain set must succeed again.
			latch(TRUE, TRUE);
			ASSERT(NOT latch.Q1);
			latch(TRUE, FALSE);
			ASSERT(latch.Q1, 'RS must set normally after a dominant reset');
			latch(FALSE, FALSE);
			ASSERT(latch.Q1, 'and hold it');
		END_FUNCTION

		{test}
		FUNCTION test_sr_toggle_sequence
			VAR
				latch: SR;
			END_VAR
			latch(TRUE, FALSE);
			latch(FALSE, TRUE);
			latch(TRUE, FALSE);
			latch(FALSE, FALSE);
			ASSERT(latch.Q1, 'set-reset-set-idle ends set');
		END_FUNCTION

		// -- SEMA -----------------------------------------------------

		{test}
		FUNCTION test_sema_first_claim_not_busy
			VAR
				sem: SEMA;
			END_VAR
			sem(CLAIM := TRUE, RELEASE := FALSE);
			ASSERT(NOT sem.BUSY, 'first claimant sees the semaphore free');
		END_FUNCTION

		{test}
		FUNCTION test_sema_second_claim_busy
			VAR
				sem: SEMA;
			END_VAR
			sem(CLAIM := TRUE, RELEASE := FALSE);
			sem(CLAIM := TRUE, RELEASE := FALSE);
			ASSERT(sem.BUSY, 'a taken semaphore reports BUSY');
		END_FUNCTION

		{test}
		FUNCTION test_sema_release_frees
			VAR
				sem: SEMA;
			END_VAR
			sem(CLAIM := TRUE, RELEASE := FALSE);
			sem(CLAIM := FALSE, RELEASE := TRUE);
			ASSERT(NOT sem.BUSY, 'released semaphore is not BUSY');
			sem(CLAIM := TRUE, RELEASE := FALSE);
			ASSERT(NOT sem.BUSY, 'and can be claimed again');
		END_FUNCTION

		{test}
		FUNCTION test_sema_claim_wins
			VAR
				sem: SEMA;
			END_VAR
			sem(CLAIM := TRUE, RELEASE := TRUE);
			sem(CLAIM := TRUE, RELEASE := FALSE);
			ASSERT(sem.BUSY, 'simultaneous claim and release: claim wins');
		END_FUNCTION
	END_NAMESPACE
END_NAMESPACE

(* ---- Console.st ---- *)
/*
The host's standard output and standard error.

`STDOUT` and `STDERR` write a `STRING` as it holds it, with no line break
added: end the text with `$N` for one. A rising edge of `REQ` writes `IN`,
once. `BUSY` is TRUE while the host takes it, and `DONE` in the call where
it has all of it, or at once for an empty text. A rising edge while `BUSY`
is ignored, as a block with `REQ` and `BUSY` ignores one: check `BUSY`
before asking again. `ERROR` is TRUE when the host has let go of its end:
the output stays closed, and each later request is an error at once. Why
the host let go is not kept.

Each block writes through a stream of bytes of its own, which it makes at
its first request and keeps, as WASI's
[standard output and error](https://github.com/WebAssembly/WASI/blob/main/proposals/cli/README.md)
take one. Two blocks hand the host two streams: the text of one comes out in
its order, but a text the host takes in parts can have the other block's
text land between them. `IN` holds 4096 bytes, and a longer `STRING` is cut
there, as any input is.

A scan never waits for the host. What it does not take within the call it
takes at later calls, while `BUSY` stays TRUE.
*/
NAMESPACE Std.Console

	/* The blocks reach WASI through what rk-bindgen writes in `generated/`
	   from WASI's WIT: each output's `WRITE_VIA_STREAM_WRITER`, in
	   `Wasi.Cli.Stdout` and in `Wasi.Cli.Stderr`, makes a stream of bytes,
	   hands its reading end to the host's `write-via-stream` and writes to
	   it. The error code the host answers with is not passed on: a write
	   only sees that the host let go. */

	/* Writes `IN` to the host's standard output on a rising edge of `REQ`.

	   # Examples

	   ```iecst
	   VAR
	       log: STDOUT;
	   END_VAR

	   log(REQ := pump_on, IN := 'pump started$N');
	   ```
	*/
	FUNCTION_BLOCK STDOUT
		VAR_INPUT
			REQ: BOOL;
			IN: STRING[4096];
		END_VAR
		VAR_OUTPUT
			BUSY: BOOL;
			DONE: BOOL;
			ERROR: BOOL;
		END_VAR
		VAR
			output: Wasi.Cli.Stdout.WRITE_VIA_STREAM_WRITER;
		END_VAR

		output(REQ := REQ, IN := IN, CLOSE := FALSE);
		BUSY := output.BUSY;
		DONE := output.DONE;
		ERROR := output.ERROR;
	END_FUNCTION_BLOCK

	/* Writes `IN` to the host's standard error on a rising edge of `REQ`.

	   # Examples

	   ```iecst
	   VAR
	       alarm: STDERR;
	   END_VAR

	   alarm(REQ := pressure > 3.0, IN := 'pressure out of range$N');
	   ```
	*/
	FUNCTION_BLOCK STDERR
		VAR_INPUT
			REQ: BOOL;
			IN: STRING[4096];
		END_VAR
		VAR_OUTPUT
			BUSY: BOOL;
			DONE: BOOL;
			ERROR: BOOL;
		END_VAR
		VAR
			output: Wasi.Cli.Stderr.WRITE_VIA_STREAM_WRITER;
		END_VAR

		output(REQ := REQ, IN := IN, CLOSE := FALSE);
		BUSY := output.BUSY;
		DONE := output.DONE;
		ERROR := output.ERROR;
	END_FUNCTION_BLOCK

	NAMESPACE Test
		USING Std.Unit;

		{test}
		FUNCTION_BLOCK test_stdout_takes_a_text
			VAR_OUTPUT
				DONE: BOOL;
			END_VAR
			VAR
				out: STDOUT;
			END_VAR
			out(REQ := TRUE, IN := 'Std.Console writes to stdout$N');
			ASSERT(NOT out.ERROR, 'STDOUT failed');
			DONE := out.DONE;
		END_FUNCTION_BLOCK

		{test}
		FUNCTION_BLOCK test_stderr_takes_a_text
			VAR_OUTPUT
				DONE: BOOL;
			END_VAR
			VAR
				err: STDERR;
			END_VAR
			err(REQ := TRUE, IN := 'Std.Console writes to stderr$N');
			ASSERT(NOT err.ERROR, 'STDERR failed');
			DONE := err.DONE;
		END_FUNCTION_BLOCK

		{test}
		FUNCTION_BLOCK test_an_empty_text_is_done_at_once
			VAR_OUTPUT
				DONE: BOOL;
			END_VAR
			VAR
				out: STDOUT;
			END_VAR
			out(REQ := TRUE, IN := '');
			ASSERT(out.DONE AND NOT out.BUSY AND NOT out.ERROR, 'an empty text was not done at once');
			DONE := TRUE;
		END_FUNCTION_BLOCK

		{test}
		FUNCTION_BLOCK test_each_rising_edge_writes_once
			VAR_OUTPUT
				DONE: BOOL;
			END_VAR
			VAR
				out: STDOUT;
				step: INT;
			END_VAR
			IF step = 0 THEN
				// The first text, until the host has all of it.
				out(REQ := TRUE, IN := 'one, ');
				ASSERT(NOT out.ERROR, 'STDOUT failed');
				IF out.DONE THEN
					step := 1;
				END_IF;
			ELSIF step = 1 THEN
				// REQ held: no second write.
				out(REQ := TRUE, IN := 'not written');
				ASSERT(NOT out.DONE AND NOT out.BUSY, 'REQ held wrote again');
				out(REQ := FALSE, IN := '');
				step := 2;
			ELSE
				// A new edge writes the second text.
				out(REQ := TRUE, IN := 'two$N');
				ASSERT(NOT out.ERROR, 'STDOUT failed');
				DONE := out.DONE;
			END_IF;
		END_FUNCTION_BLOCK
	END_NAMESPACE
END_NAMESPACE
